FUNCTION Fun_CalculoCoordenadasFinalesFormacion : bool
VAR_INPUT
	TipoCalForCavallete 		: UINT ;
	numeroLastre_int 		: UINT ;
	Supporto 				: POINTER TO TFMachinePalletizer_Pallet;
	XFinale 				: POINTER TO  ARRAY [1..MAXFORMINGSLAB] OF LREAL;
	YFinale 				: POINTER TO  ARRAY [1..MAXFORMINGSLAB] OF LREAL;
	YInternoLastra 			: POINTER TO  ARRAY [1..MAXFORMINGSLAB] OF LREAL;
	ZFinale 				: POINTER TO  ARRAY [1..MAXFORMINGSLAB] OF LREAL;
	ZInternoLastra			: POINTER TO  ARRAY [1..MAXFORMINGSLAB] OF LREAL;
	JFinale 				: POINTER TO  ARRAY [1..MAXFORMINGSLAB] OF LREAL;
END_VAR
VAR
	Contador: UINT;
END_VAR

FOR Contador := 1 TO numeroLastre_int * 2 DO 
	CASE TipoCalForCavallete OF 
		1: 

			XFinale^[Contador] := Supporto^.XDim/2 + Supporto^.OFSDE_X180;
			;
		2: 
			;
		3:
			;
		4: 
			;
	END_CASE
	
END_FOR

END_FUNCTION

(* stored: Version 1.1.0.1, ProductVersion 3.1.4024.11
   POU Fun_CalculoCoordenadasFinalesFormacion: Id {3f8db5d7-85e7-4ed0-803f-96d110a21ee7}, SpecialFunc None *)
